// TIA Portal project "Step7" (V20)

(* hardware
DEVICE "S120Democase"  SINAMICS S120
   slot 0: "S120Democase"  S120 CU320-2 PN  6SL3040-1MA01-0Axx  V5.2.3
      slot 1: "PROFINET interface"  PROFINET
      slot 3: "Ethernet commissioning interface"  LAN
   slot 0: "Drive control"  S120 CU320-2 PN
   slot 1: "TB30"  TB
      slot 500: "TB30"  TB30  6SL3055-0AA00-2Txx
   slot 2: "RedAxis"  DMM
      slot 200: "DMM"  RedAxis  6SL3120-2TE13-0Axx
      slot 300: "Encoder evaluation_1"  RedAxis  1FK7022-xAK7x-xLGx
      slot 400: "Measuring system_1"  RedAxis  1FK7022-xAK7x-xLGx
      slot 1000: "RedMotor_X1"  RedAxis  1FK7022-xAK7x-xLGx
   slot 3: "BlueAxis"  DMM
      slot 200: "Motor Module_1"  BlueAxis  6SL3120-2TE13-0Axx
      slot 300: "Encoder evaluation_1"  BlueAxis  xxxxxxx-xxxxx-xxxx
      slot 400: "Measuring system_1"  BlueAxis  1FK7022-xAK71-xAGx
      slot 1000: "BlueMotor_X2"  BlueAxis  1FK7022-xAK71-xAGx
DEVICE "PLC_S120Democase"  S7-1500 station
   slot 0: "Rail_0"  Rack  6ES7 590-1***0-0AA0
   slot 1: "PLC_S120Democase"  CPU 1515TF-2 PN  6ES7 515-2UM01-0AB0  V2.9
      slot 3: "CPU display_1"  6ES7591-1BA00-0AA0
      slot 32768: "PROFINET interface_1"  X1
         slot 32769: "Port_1"  X1 P1
         slot 32770: "Port_2"  X1 P2
      slot 33024: "PROFINET interface_2"  X2
         slot 33025: "Port_1"  X2 P1
      slot 34817: "Virtual CP interface port_1"  Virtual CP interface port  Virtual CP interface port
DEVICE "PLC_1"  S7-1500 station
   slot 0: "Rail_0"  Rack  6ES7 590-1***0-0AA0
   slot 1: "PLC_1"  CPU 1515TF-2 PN  6ES7 515-2UN03-0AB0  V4.0
      slot 3: "CPU display_1"  6ES7591-1BA00-0AA0
      slot 32768: "PROFINET interface_1"  X1
         slot 32769: "Port_1"  X1 P1
         slot 32770: "Port_2"  X1 P2
      slot 33024: "PROFINET interface_2"  X2
         slot 33025: "Port_1"  X2 P1
      slot 34817: "Virtual CP interface port_1"  Virtual CP interface port  Virtual CP interface port FW V4.0
DEVICE "PLC_2"  S7-1500 station
   slot 0: "Rail_0"  Rack  6ES7 590-1***0-0AA0
   slot 1: "PLC_2"  CPU 1515TF-2 PN  6ES7 515-2UN03-0AB0  V4.0
      slot 3: "CPU display_1"  6ES7591-1BA00-0AA0
      slot 32768: "PROFINET interface_1"  X1
         slot 32769: "Port_1"  X1 P1
         slot 32770: "Port_2"  X1 P2
      slot 33024: "PROFINET interface_2"  X2
         slot 33025: "Port_1"  X2 P1
      slot 34817: "Virtual CP interface port_1"  Virtual CP interface port  Virtual CP interface port FW V4.0
*)

// ===== PLC "PLC_S120Democase"  CPU 1515TF-2 PN =====

VAR_GLOBAL   // PLC tag table "Default tag table"
   "SynchronousAxis_red_Actor_Interface_AddressIn" AT %I260.0 : "PD_TEL105_IN";
   "SynchronousAxis_red_Actor_Interface_AddressOut" AT %Q260.0 : "PD_TEL105_OUT";
   "PositioningAxis_blue_Actor_Interface_AddressIn" AT %I280.0 : "PD_TEL105_IN";
   "PositioningAxis_blue_Actor_Interface_AddressOut" AT %Q280.0 : "PD_TEL105_OUT";
   "Clock_Byte" AT %MB0 : Byte;
   "Clock_10Hz" AT %M0.0 : Bool;
   "Clock_5Hz" AT %M0.1 : Bool;
   "Clock_2.5Hz" AT %M0.2 : Bool;
   "Clock_2Hz" AT %M0.3 : Bool;
   "Clock_1.25Hz" AT %M0.4 : Bool;
   "Clock_1Hz" AT %M0.5 : Bool;
   "Clock_0.625Hz" AT %M0.6 : Bool;
   "Clock_0.5Hz" AT %M0.7 : Bool;
END_VAR

VAR_GLOBAL   // PLC tag table "DemocaseAppTagTable"
   "ControlUnit_AddressIn" AT %I300.0 : "PD_TEL_393_IN";
   "ControlUnit_AddressOut" AT %Q300.0 : "PD_TEL_393_OUT";
   "ET200_AI_0" AT %IW2 : Int;
   "ET200_AI_1" AT %IW4 : Int;
   "OutputCam_1_Interface_Address" AT %Q303.5 : Bool;
   "TB30_AI_0" AT %IW342 : Word;
   "TB30_AI_1" AT %IW344 : Word;
END_VAR

TYPE "PD_TEL_393_IN"
   STRUCT
      CU_ZSW1 : Struct
         Bit_08 : Bool;
         Bit_09 : Bool;
         Bit_10 : Bool;
         Bit_11 : Bool;
         Bit_12 : Bool;
         Bit_13 : Bool;
         Bit_14 : Bool;
         Bit_15 : Bool;
         Bit_00 : Bool;
         Bit_01 : Bool;
         Bit_02 : Bool;
         Bit_03 : Bool;
         Bit_04 : Bool;
         Bit_05 : Bool;
         Bit_06 : Bool;
         Bit_07 : Bool;
      END_STRUCT;
      E_DIGITAL : Struct
         DI_00 : Bool;   // Switch 0
         DI_01 : Bool;   // Switch 1
         DI_02 : Bool;   // Switch 2
         DI_03 : Bool;   // Switch 3
         DI_04 : Bool;   // Switch 4
         DI_05 : Bool;   // Switch 5
         DI_06 : Bool;   // Switch 6
         DI_07 : Bool;   // Switch 7
         DIDO_08 : Bool;   // Switch 8
         DIDO_09 : Bool;   // Switch 9
         DIDO_10 : Bool;   // Switch 10
         DIDO_11 : Bool;   // Switch 11
         DIDO_12 : Bool;   // Switch 12
         DIDO_13 : Bool;   // Switch 13
         DIDO_14 : Bool;
         DIDO_15 : Bool;
      END_STRUCT;
      E_DIGITAL_1 : Struct
         DI_16 : Bool;
         DI_17 : Bool;   // SafeHold switch
         DI_18 : Bool;   // InfeedReady
         DI_19 : Bool;
         DI_20 : Bool;   // Switch 14
         DI_21 : Bool;   // Switch 15
         DI_22 : Bool;
         Bit_07 : Bool;
         Bit_08 : Bool;
         Bit_09 : Bool;
         Bit_10 : Bool;
         Bit_11 : Bool;
         Bit_12 : Bool;
         Bit_13 : Bool;
         Bit_14 : Bool;
         Bit_15 : Bool;
      END_STRUCT;
      MT_ZTW : Word;
      MT1_ZS_F : Word;
      MT1_ZS_S : Word;
      MT2_ZS_F : Word;
      MT2_ZS_S : Word;
      MT3_ZS_F : Word;
      MT3_ZS_S : Word;
      MT4_ZS_F : Word;
      MT4_ZS_S : Word;
      MT5_ZS_F : Word;
      MT5_ZS_S : Word;
      MT6_ZS_F : Word;
      MT6_ZS_S : Word;
      MT7_ZS_F : Word;
      MT7_ZS_S : Word;
      MT8_ZS_F : Word;
      MT8_ZS_S : Word;
      E_ANALOG : Word;
   END_STRUCT;
END_TYPE

TYPE "PD_TEL_393_OUT"
   STRUCT
      CU_STW : Struct
         Bit_08 : Bool;
         Bit_09 : Bool;
         Bit_10 : Bool;
         Bit_11 : Bool;
         Bit_12 : Bool;
         Bit_13 : Bool;
         Bit_14 : Bool;
         Bit_15 : Bool;
         Bit_00 : Bool;
         Bit_01 : Bool;
         Bit_02 : Bool;
         Bit_03 : Bool;
         Bit_04 : Bool;
         Bit_05 : Bool;
         Bit_06 : Bool;
         Acknowledge : Bool;
      END_STRUCT;
      A_DIGITAL : Struct
         DIO_08 : Bool;
         DIO_09 : Bool;
         DIO_10 : Bool;
         DIO_11 : Bool;
         DIO_12 : Bool;
         DIO_13 : Bool;
         DIO_14 : Bool;
         DIO_15 : Bool;
         Bit_00 : Bool;
         Bit_01 : Bool;
         Bit_02 : Bool;
         Bit_03 : Bool;
         Bit_04 : Bool;
         Bit_05 : Bool;
         Bit_06 : Bool;
         Bit_07 : Bool;
      END_STRUCT;
      A_DIGITAL_1 : Struct
         Bit_08 : Bool;
         Bit_09 : Bool;
         Bit_10 : Bool;
         Bit_11 : Bool;
         Bit_12 : Bool;
         Bit_13 : Bool;
         Bit_14 : Bool;
         Bit_15 : Bool;
         DIO_16 : Bool;
         Bit_01 : Bool;
         Bit_02 : Bool;
         Bit_03 : Bool;
         Bit_04 : Bool;
         Bit_05 : Bool;
         Bit_06 : Bool;
         Bit_07 : Bool;
      END_STRUCT;
      MT_STW : Struct
         Bit_08 : Bool;
         Bit_09 : Bool;
         Bit_10 : Bool;
         Bit_11 : Bool;
         Bit_12 : Bool;
         Bit_13 : Bool;
         Bit_14 : Bool;
         Bit_15 : Bool;
         Bit_16 : Bool;
         Bit_00 : Bool;
         Bit_01 : Bool;
         Bit_02 : Bool;
         Bit_03 : Bool;
         Bit_04 : Bool;
         Bit_05 : Bool;
         Bit_06 : Bool;
         Bit_07 : Bool;
      END_STRUCT;
   END_STRUCT;
END_TYPE

DATA_BLOCK "Main_Safety_RTG1_DB"   // DB1, F_DB
{ S7_Optimized_Access := 'TRUE' }
NAME : FUSI
VERSION : 0.1
// stored: InstanceOfName Main_Safety_RTG1
"Main_Safety_RTG1"
BEGIN
END_DATA_BLOCK

DATA_BLOCK "GlobalBlock"   // DB2
{ S7_Optimized_Access := 'TRUE' }
VERSION : 0.1
BEGIN
END_DATA_BLOCK

DATA_BLOCK "Axis_blue_DB"   // DB10
{ S7_Optimized_Access := 'TRUE' }
VERSION : 0.1
// stored: InstanceOfName Axis_blue
"Axis_blue"
BEGIN
END_DATA_BLOCK

DATA_BLOCK "Axis_red_DB"   // DB11
{ S7_Optimized_Access := 'TRUE' }
VERSION : 0.1
// stored: InstanceOfName Axis_red
"Axis_red"
BEGIN
END_DATA_BLOCK

DATA_BLOCK "PositioningAxis_blue"   // DB4, Motion_DB
{ S7_Optimized_Access := 'TRUE' }
AUTHOR : SIMATIC
FAMILY : MC_1500
VERSION : 6.0
// stored: InstanceOfName TO_PositioningAxis
"TO_PositioningAxis"
BEGIN
END_DATA_BLOCK

DATA_BLOCK "SynchronousAxis_red"   // DB6, Motion_DB
{ S7_Optimized_Access := 'TRUE' }
AUTHOR : SIMATIC
FAMILY : MC_1500
VERSION : 6.0
// stored: InstanceOfName TO_SynchronousAxis
"TO_SynchronousAxis"
BEGIN
END_DATA_BLOCK

FUNCTION_BLOCK "Main_Safety_RTG1"   // FB1, F_FBD
{ S7_Optimized_Access := 'TRUE' }
BEGIN
END_FUNCTION_BLOCK

FUNCTION_BLOCK "SclBlock"   // FB2, SCL
{ S7_Optimized_Access := 'TRUE' }
VERSION : 0.1
BEGIN
END_FUNCTION_BLOCK

FUNCTION_BLOCK "Axis_blue"   // FB10, FBD
{ S7_Optimized_Access := 'TRUE' }
VERSION : 0.1
// FB for the blue axis
   VAR
      MC_POWER_Instance : MC_POWER;
      MC_RESET_Instance : MC_RESET;
      MC_HOME_Instance : MC_HOME;
      MC_HALT_Instance : MC_HALT;
      MC_MOVEVELOCITY_Instance : MC_MOVEVELOCITY;
      MC_MOVERELATIVE_Instance : MC_MOVERELATIVE;
      MC_MOVEABSOLUTE_Instance : MC_MOVEABSOLUTE;
      MC_OUTPUTCAM_Instance : MC_OUTPUTCAM;
   END_VAR
   VAR_TEMP
      tempVelocity : LReal;
      velocity : LReal;
   END_VAR
BEGIN

REGION Network 1
   // Call basic MotionControl commands
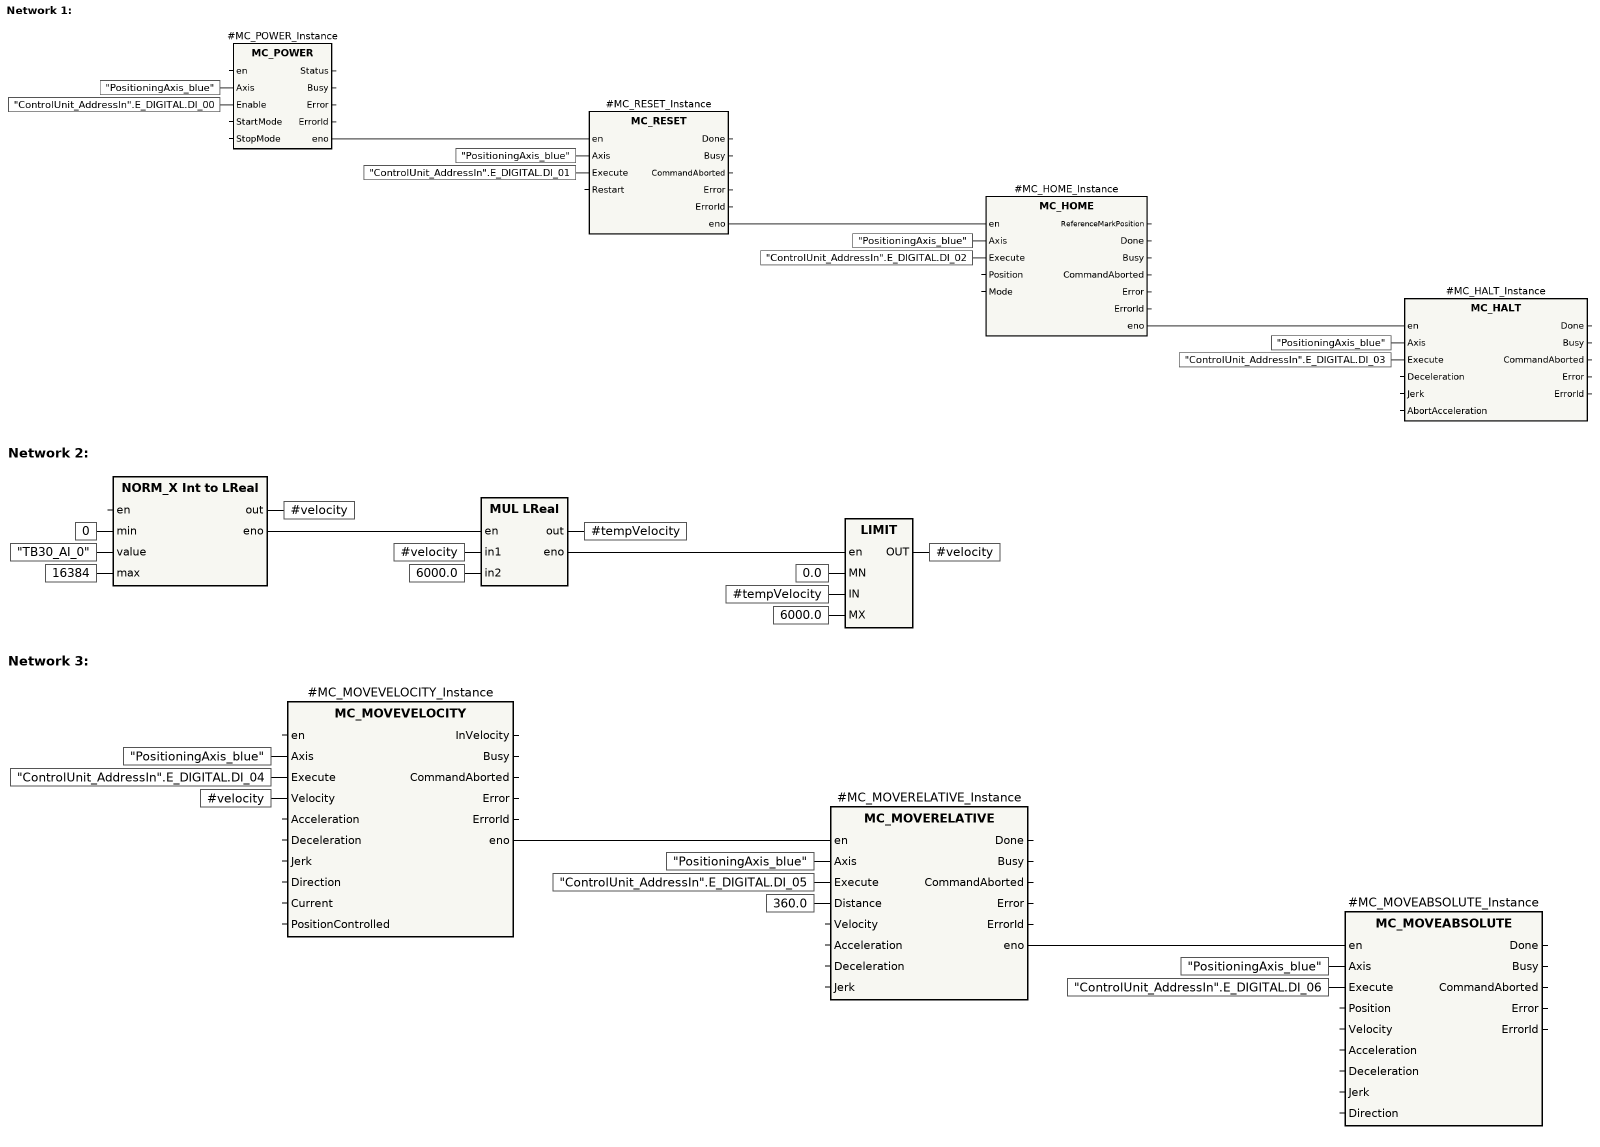
   // ENO of a box is taken as its EN; it also drops when the box reports an error
   #MC_POWER_Instance(Axis := "PositioningAxis_blue", Enable := "ControlUnit_AddressIn".E_DIGITAL.DI_00);   // MC_POWER
   #MC_RESET_Instance(Axis := "PositioningAxis_blue", Execute := "ControlUnit_AddressIn".E_DIGITAL.DI_01);   // MC_RESET
   #MC_HOME_Instance(Axis := "PositioningAxis_blue", Execute := "ControlUnit_AddressIn".E_DIGITAL.DI_02);   // MC_HOME
   #MC_HALT_Instance(Axis := "PositioningAxis_blue", Execute := "ControlUnit_AddressIn".E_DIGITAL.DI_03);   // MC_HALT: MC_Halt is used (and not MC_Stop) because it just stops an axis, without lockking it.
END_REGION

REGION Network 2
   // Read in analoge value and create setpoint (0 to 6000 °/s) = (0 rpm tp +1000 rpm)
   #velocity := NORM_X(MIN := 0, VALUE := "TB30_AI_0", MAX := 16384);
   #tempVelocity := #velocity * 6000.0;
   #velocity := LIMIT(MN := 0.0, IN := #tempVelocity, MX := 6000.0);
END_REGION

REGION Network 3
   // MotionControl commands for the blue axis
   // ENO of a box is taken as its EN; it also drops when the box reports an error
   #MC_MOVEVELOCITY_Instance(Axis := "PositioningAxis_blue",   // MC_MOVEVELOCITY
                           Execute := "ControlUnit_AddressIn".E_DIGITAL.DI_04,
                           Velocity := #velocity);
   #MC_MOVERELATIVE_Instance(Axis := "PositioningAxis_blue",   // MC_MOVERELATIVE
                           Execute := "ControlUnit_AddressIn".E_DIGITAL.DI_05,
                           Distance := 360.0);
   #MC_MOVEABSOLUTE_Instance(Axis := "PositioningAxis_blue", Execute := "ControlUnit_AddressIn".E_DIGITAL.DI_06);   // MC_MOVEABSOLUTE
END_REGION
END_FUNCTION_BLOCK

FUNCTION_BLOCK "Axis_red"   // FB11, FBD
{ S7_Optimized_Access := 'TRUE' }
VERSION : 0.1
// FB for the red axis
   VAR
      MC_POWER_Instance : MC_POWER;
      MC_RESET_Instance : MC_RESET;
      MC_HOME_Instance : MC_HOME;
      MC_HALT_Instance : MC_HALT;
      MC_MOVEVELOCITY_Instance : MC_MOVEVELOCITY;
      MC_GEARIN_Instance : MC_GEARIN;
      MC_MOVERELATIVE_1 : MC_MOVERELATIVE;
   END_VAR
BEGIN

REGION Network 1
   // Call basic MotionControl commands
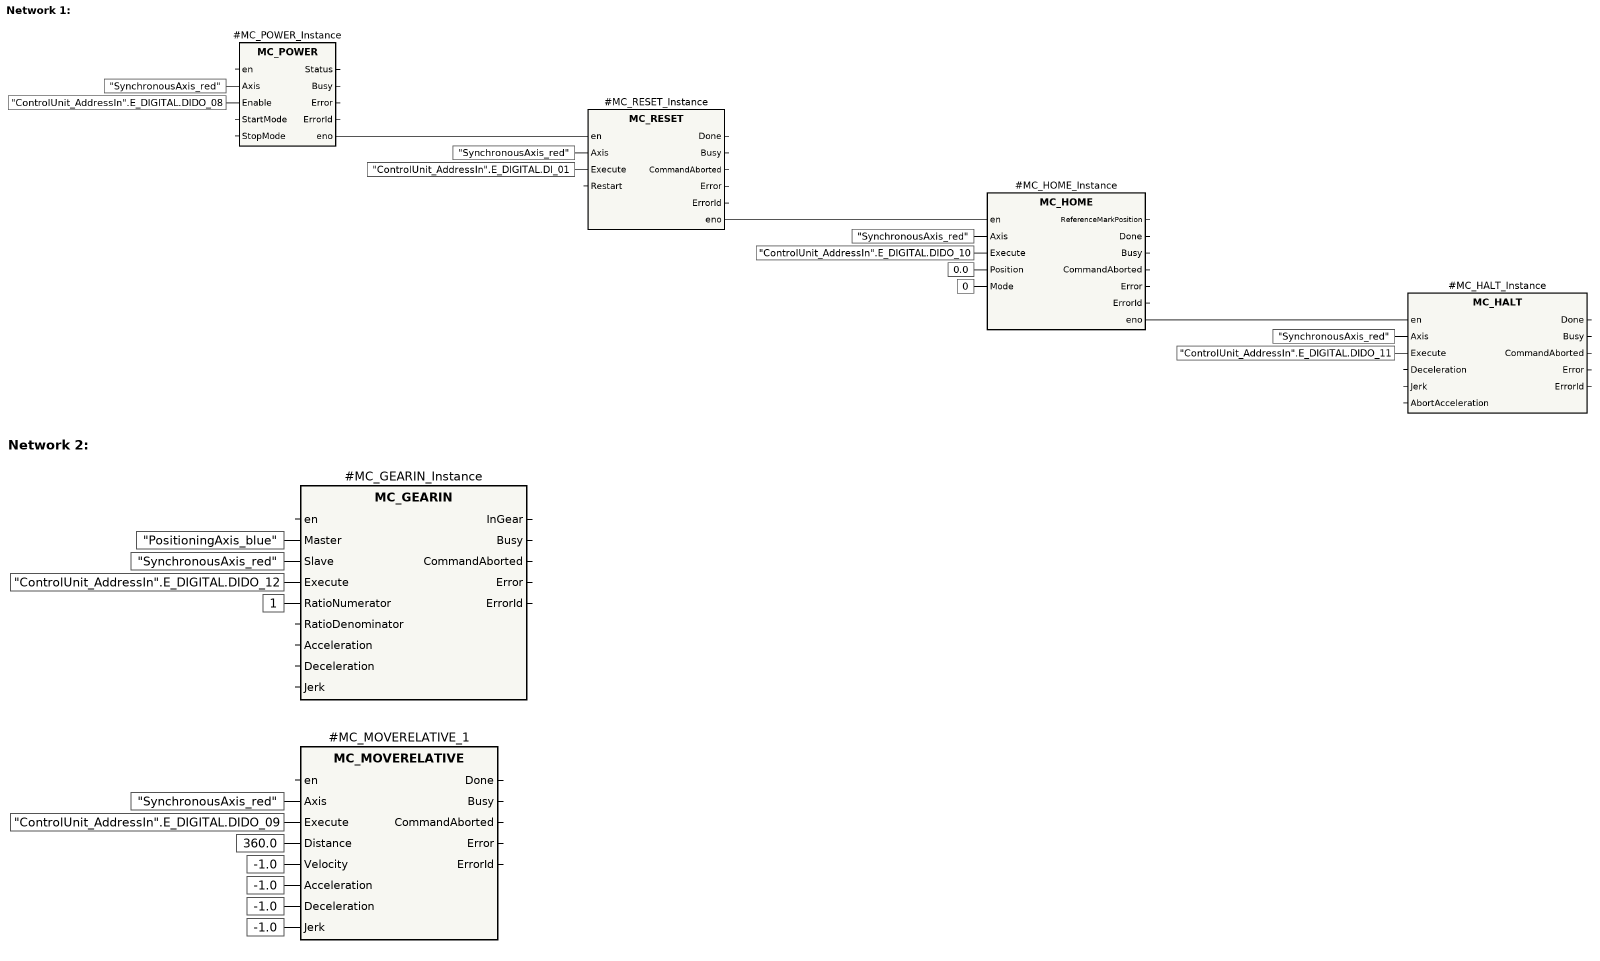
   // ENO of a box is taken as its EN; it also drops when the box reports an error
   #MC_POWER_Instance(Axis := "SynchronousAxis_red", Enable := "ControlUnit_AddressIn".E_DIGITAL.DIDO_08);   // MC_POWER
   #MC_RESET_Instance(Axis := "SynchronousAxis_red", Execute := "ControlUnit_AddressIn".E_DIGITAL.DI_01);   // MC_RESET
   #MC_HOME_Instance(Axis := "SynchronousAxis_red",   // MC_HOME
                     Execute := "ControlUnit_AddressIn".E_DIGITAL.DIDO_10,
                     Position := 0.0,
                     Mode := 0);
   #MC_HALT_Instance(Axis := "SynchronousAxis_red", Execute := "ControlUnit_AddressIn".E_DIGITAL.DIDO_11);   // MC_HALT: MC_Halt is used (and not MC_Stop) because it just stops an axis, without lockking it.
END_REGION

REGION Network 2
   // MotionControl commands for the red axis
   #MC_GEARIN_Instance(Master := "PositioningAxis_blue",   // MC_GEARIN
                       Slave := "SynchronousAxis_red",
                       Execute := "ControlUnit_AddressIn".E_DIGITAL.DIDO_12,
                       RatioNumerator := 1);
   #MC_MOVERELATIVE_1(Axis := "SynchronousAxis_red",   // MC_MOVERELATIVE
                      Execute := "ControlUnit_AddressIn".E_DIGITAL.DIDO_09,
                      Distance := 360.0,
                      Velocity := -1.0,
                      Acceleration := -1.0,
                      Deceleration := -1.0,
                      Jerk := -1.0);
END_REGION

REGION Network 3
   // Move commands
END_REGION
END_FUNCTION_BLOCK

ORGANIZATION_BLOCK "Main"   // OB1, LAD, ProgramCycle
TITLE = "Main Program Sweep (Cycle)"
{ S7_Optimized_Access := 'TRUE' }
VERSION : 0.1
   VAR_INPUT
      Initial_Call : Bool;   // Initial call of this OB
      Remanence : Bool;   // =True, if remanent data are available
   END_VAR
BEGIN
END_ORGANIZATION_BLOCK

ORGANIZATION_BLOCK "DriveController_Main"   // OB123, LAD, ProgramCycle
TITLE = "Main Program Sweep (Cycle)"
{ S7_Optimized_Access := 'TRUE' }
VERSION : 0.1
   VAR_INPUT
      Initial_Call : Bool;   // Initial call of this OB
      Remanence : Bool;   // =True, if remanent data are available
   END_VAR
BEGIN

REGION Network 1
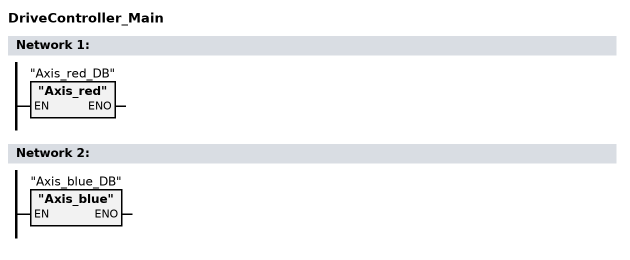
   RUNG wire#powerrail
      "Axis_red_DB"()
   END_RUNG
   // the same network as SCL:
   "Axis_red_DB"();   // "Axis_red"
END_REGION

REGION Network 2
   RUNG wire#powerrail
      "Axis_blue_DB"()
   END_RUNG
   // the same network as SCL:
   "Axis_blue_DB"();   // "Axis_blue"
END_REGION
END_ORGANIZATION_BLOCK

// ===== PLC "PLC_1"  CPU 1515TF-2 PN =====

DATA_BLOCK "Main_Safety_RTG1_DB"   // DB1, F_DB
{ S7_Optimized_Access := 'TRUE' }
NAME : FUSI
VERSION : 0.1
// stored: InstanceOfName Main_Safety_RTG1
"Main_Safety_RTG1"
BEGIN
END_DATA_BLOCK

FUNCTION_BLOCK "Main_Safety_RTG1"   // FB1, F_FBD
{ S7_Optimized_Access := 'TRUE' }
BEGIN
END_FUNCTION_BLOCK

ORGANIZATION_BLOCK "Main"   // OB1, LAD, ProgramCycle
TITLE = "Main Program Sweep (Cycle)"
{ S7_Optimized_Access := 'TRUE' }
VERSION : 0.1
   VAR_INPUT
      Initial_Call : Bool;   // Initial call of this OB
      Remanence : Bool;   // =True, if remanent data are available
   END_VAR
BEGIN
END_ORGANIZATION_BLOCK

// ===== PLC "PLC_2"  CPU 1515TF-2 PN =====

DATA_BLOCK "Main_Safety_RTG1_DB"   // DB1, F_DB
{ S7_Optimized_Access := 'TRUE' }
NAME : FUSI
VERSION : 0.1
// stored: InstanceOfName Main_Safety_RTG1
"Main_Safety_RTG1"
BEGIN
END_DATA_BLOCK

FUNCTION_BLOCK "Main_Safety_RTG1"   // FB1, F_FBD
{ S7_Optimized_Access := 'TRUE' }
BEGIN
END_FUNCTION_BLOCK

ORGANIZATION_BLOCK "Main"   // OB1, LAD, ProgramCycle
TITLE = "Main Program Sweep (Cycle)"
{ S7_Optimized_Access := 'TRUE' }
VERSION : 0.1
   VAR_INPUT
      Initial_Call : Bool;   // Initial call of this OB
      Remanence : Bool;   // =True, if remanent data are available
   END_VAR
BEGIN
END_ORGANIZATION_BLOCK